{attribute 'linkalways'} 
{attribute 'no_explicit_call' := 'This FB is a CLASS and must be accessed using methods or properties'}
{attribute 'enable_dynamic_creation'}
FUNCTION_BLOCK _ETcVnFlipAxis EXTENDS EnumDatatypeBase
VAR
	localData : ETcVnFlipAxis;
	activeData : REFERENCE TO ETcVnFlipAxis;
	enumBaseDatatype : _INT(localData);
END_VAR

METHOD PRIVATE AddLocalEnumeration
VAR_INPUT
	Enumeration : T_MAXSTRING;
	Value : ETcVnFlipAxis;
END_VAR
AddEnumeration(Enumeration, Value);
END_METHOD

PROPERTY PUBLIC Address : PVOID
GET
Address := ADR(activeData);
END_GET
END_PROPERTY

METHOD PUBLIC ClearReference
VAR_INPUT
END_VAR
activeData REF= localData;
SetBaseDatatypeReference();
END_METHOD

METHOD PUBLIC Clone : I_Datatype
VAR
    pClone : POINTER TO _ETcVnFlipAxis;
END_VAR
pClone := __NEW(_ETcVnFlipAxis(InitialValue := Value));
Clone := pClone^;
END_METHOD

METHOD FB_init : BOOL
VAR_INPUT
	bInitRetains : BOOL; // if TRUE, the retain variables are initialized (warm start / cold start)
	bInCopyCode : BOOL;  // if TRUE, the instance afterwards gets moved into the copy code (online change)
	InitialValue : ETcVnFlipAxis;
END_VAR
localData := InitialValue;
AddBaseDatatype(enumBaseDatatype);
ClearReference();

AddLocalEnumeration('TCVN_FA_XY', ETcVnFlipAxis.TCVN_FA_XY);
AddLocalEnumeration('TCVN_FA_X', ETcVnFlipAxis.TCVN_FA_X);
AddLocalEnumeration('TCVN_FA_Y', ETcVnFlipAxis.TCVN_FA_Y);
END_METHOD

PROPERTY PUBLIC Identifier : T_MAXSTRING
GET
Identifier := 'ETcVnFlipAxis';
END_GET
END_PROPERTY

METHOD IsEnumeratorValueEqual : BOOL
VAR_INPUT
	Enumerator : I_KeyValueForwardEnumerator;
END_VAR
VAR
	storedValue : ETcVnFlipAxis;
END_VAR
IF NOT Enumerator.TryGet(storedValue) THEN
	RETURN;
END_IF

IsEnumeratorValueEqual := storedValue = activeData;
END_METHOD

METHOD PUBLIC MakeReferenceTo
VAR_INPUT
	ReferenceTarget : REFERENCE TO ETcVnFlipAxis;
END_VAR
activeData REF= ReferenceTarget;
SetBaseDatatypeReference();
END_METHOD

METHOD PROTECTED SetBaseDatatypeReference
VAR_INPUT
END_VAR
enumBaseDatatype.MakeReferenceTo(activeData);
END_METHOD

PROPERTY PUBLIC Size : UDINT
GET
Size := SIZEOF(activeData);
END_GET
END_PROPERTY

METHOD TryMakeReferenceTo : BOOL
VAR_INPUT
	Target : I_Datatype;
END_VAR
VAR
	targetAsEnum : I_EnumDatatype;
	pTargetData : POINTER TO ETcVnFlipAxis;
END_VAR
IF NOT Target.TryResolveAsEnumDatatype(targetAsEnum) THEN
	RETURN;
END_IF

IF targetAsEnum.Identifier <> Identifier THEN
	RETURN;
END_IF

pTargetData := Target.Address;
activeData REF= pTargetData^;
SetBaseDatatypeReference();
TryMakeReferenceTo := TRUE;
END_METHOD

PROPERTY PUBLIC Value : ETcVnFlipAxis
GET
Value := activeData;
END_GET
SET
activeData := Value;
END_SET
END_PROPERTY

END_FUNCTION_BLOCK

(* stored: Version 1.1.0.1
   POU _ETcVnFlipAxis: Id {7d214fab-df57-47d6-8e95-c2455749fd54}, SpecialFunc None
   Folder Constructor: Id {05c2a129-a1f4-4fac-a058-05de9a086f69}
   Folder Private: Id {a81ffb5d-786a-422c-af45-e54caaa6acf3}
   Folder Protected: Id {f324d0c5-a498-4a92-894e-3798e6e74cd3}
   Method AddLocalEnumeration: Id {32241d5c-dfe6-405d-a67c-2e8fda40d8de}
   Property Address: Id {1dc68565-e81b-43ec-8d01-d159908562ba}
   Get Get: Id {2482492c-c719-45cf-abeb-c729e1ec738c}
   Method ClearReference: Id {74fda18c-7f65-4b94-83f1-b53d838d5538}
   Method Clone: Id {9b11e133-99e8-441e-945a-2da2b35d06cb}
   Method FB_init: Id {5ffbf61f-601e-4b78-9c9b-4adb9b35c8a5}
   Property Identifier: Id {8dbfe242-99b9-4640-9c58-2097062a1320}
   Get Get: Id {f41092ec-b84a-45d9-956d-45afcc560d23}
   Method IsEnumeratorValueEqual: Id {469ec699-f7eb-4629-8728-dfb230763335}
   Method MakeReferenceTo: Id {d5d2fc38-5d59-4ad5-9bfb-3386d4f0f678}
   Method SetBaseDatatypeReference: Id {ed427fae-e2e0-406f-a953-c6bd91f653f0}
   Property Size: Id {fd10714a-499d-408b-98d1-4e3aa97542cc}
   Get Get: Id {a51f17ba-7f54-4505-bd62-a4a4940b4424}
   Method TryMakeReferenceTo: Id {a2eb400a-f51d-4c80-99d1-42c1f19dd6ae}
   Property Value: Id {47ef7db8-0f29-42fd-9881-7f019ff8b699}
   Get Get: Id {2dc2a7a8-03a9-4050-b148-2cf3d6df582b}
   Set Set: Id {550debe8-d286-4006-a2e2-8aea109d9445} *)
